// SIMATIC S7-200 project (STEP 7-Micro/WIN), CPU 224 REL 02.01

ORGANIZATION_BLOCK MAIN:OB1
TITLE=PROGRAM COMMENTS
BEGIN
Network 1 // Network Title
// Network Comment
LD     I0.0
MOVW   +250, VW0
-I     AIW8, VW0
Network 2
// (network saved uncompiled; FBD cells follow)
// row 0: c1 [SUB_I ]
// row 1: c1 [ EN:=I0.0, IN1:=0, IN2:=+2, ENO=>V?0, OUT=>VW2]
// row 2: c1 [box]
// row 3: c1 [box]
Network 3
LD     I0.0
MOVW   VW0, VW4
*I     VW2, VW4
Network 4
// (network saved uncompiled; FBD cells follow)
// row 0: c3 [MOV_W ]
// row 1: c1 [>I VW4 0 ]  c2 --  c3 [ EN:=power@row1, IN:=VW4, ENO=>V?0, OUT=>AQW0]
// row 2: c1 [box]  c3 [box]
Network 5
// (network saved uncompiled; FBD cells follow)
// row 0: c3 [MOV_W ]
// row 1: c1 [>=I 0 VW4 ]  c2 --  c3 [ EN:=power@row1, IN:=0, ENO=>V?0, OUT=>AQW0]
// row 2: c1 [box]  c3 [box]
Network 6
LDW>   VW0, 0
=      Q0.0
END_ORGANIZATION_BLOCK
